// TIA Portal V17 export
// export: Created 2026-04-13T11:12:52.9445675Z, ExportSetting WithDefaults, DisplayName Totally Integrated Automation Portal, DisplayVersion V17 Update 4, DisplayName TIA Portal Openness, DisplayVersion V17 Update 4, DisplayName TIA Portal Version Control Interface, DisplayVersion V17, DisplayName SINAMICS Startdrive Advanced, DisplayVersion V17, DisplayName SINAMICS Startdrive G130, G150, S120, S150, SINAMICS MV, S210, DisplayVersion V17, DisplayName SINAMICS Startdrive G110M, G120, G120C, G120D, G120P, G115D, DisplayVersion V17, DisplayName STEP 7 Professional, DisplayVersion V17 Update 4, DisplayName STEP 7 Safety, DisplayVersion V17, DisplayName WinCC Professional, DisplayVersion V17 Update 4
TagTable "DH"
  DH_XH循环风机动画 : Int  (PLC tag DH.XH循环风机动画, HMI_连接_1, 1 s)
  DH_JL进料泵动画 : Int  (PLC tag DH.JL进料泵动画, HMI_连接_1, 1 s)
  DH_JB搅拌电机动画 : Int  (PLC tag DH.JB搅拌电机动画, HMI_连接_1, 1 s)
  DH_主管道动画 : Int  (PLC tag DH.主管道动画, HMI_连接_1, 1 s)
  DH_YF引风机动画 : Int  (PLC tag DH.YF引风机动画, HMI_连接_1, 1 s)
  DH_SF送风机动画 : Int  (PLC tag DH.SF送风机动画, HMI_连接_1, 1 s)
  DH_LX离心雾化动画 : Int  (PLC tag DH.LX离心雾化动画, HMI_连接_1, 1 s)
